Fanuc KAREL source: compact_preamble.KL

PROGRAM IO0019
%NOLOCKGROUP
ROUTINE RTEST
VAR
L1 : ARRAY[3] OF INTEGER;L2 : XYZWPR
L3 : JOINTPOS9
L4 : POSITION
A:BOOLEAN
B:REAL
C:REAL
D:BOOLEAN
E:REAL
BEGIN
A=TRUE
L1[1]=2
D=TRUE
E=1.0
DOUT[1]=TRUE
END RTEST
BEGIN
RTEST
END IO0019
